// TIA Portal V17 export
// export: Created 2025-06-20T10:23:48.7607854Z, ExportSetting WithDefaults, DisplayName Totally Integrated Automation Portal, DisplayVersion V17 Update 8, DisplayName TIA Portal Openness, DisplayVersion V17 Update 8, DisplayName TIA Portal Version Control Interface, DisplayVersion V17, DisplayName SINAMICS Startdrive Advanced, DisplayVersion V17 SP2, DisplayName SINAMICS Startdrive G110M, G120, G120C, G120D, G120P, G115D, DisplayVersion V17 SP2, DisplayName SINAMICS Startdrive G130, G150, S120, S150, SINAMICS MV, S210, DisplayVersion V17 SP2, DisplayName STEP 7 Professional, DisplayVersion V17 Update 8, DisplayName SINUMERIK ONE STEP 7 Toolbox, DisplayVersion V17 Update 12, DisplayName SINUMERIK ONE PLC Basic Program Plus, DisplayVersion V17 Update 12, DisplayName SINUMERIK 840D sl STEP 7 Toolbox, DisplayVersion V17 Update 12, DisplayName STEP 7 Safety, DisplayVersion V17 Update 6, DisplayName WinCC Advanced, DisplayVersion V17 Update 8
FUNCTION "FC441_MACHINE_POWDER_ALARM_DECODING" : Void   // FC441, LAD
{ S7_Optimized_Access := 'FALSE' }
AUTHOR : ETXETAR
VERSION : 1.0
// stored: AutoNumber false, IsIECCheckEnabled false, SetENOAutomatically false, UDAEnableTagReadback false
   VAR_TEMP
      RST_ALARMS_1 : Bool;   // RESET ALARMS 1
      RST_ALARMS_2 : Bool;   // RESET ALARMS 2
      ZERO : Int;   // ZERO
      RET_VAL_1 : Int;   // RET VALUE
   END_VAR
   VAR CONSTANT
      FC_CONSTANT : Int := 440;
   END_VAR
   VAR_TEMP   // added for the SCL form of the ladder/FBD networks
      _w1 : Bool;
      _w2 : Bool;
      _w3 : Bool;
   END_VAR
BEGIN

REGION Network 1: ZERO
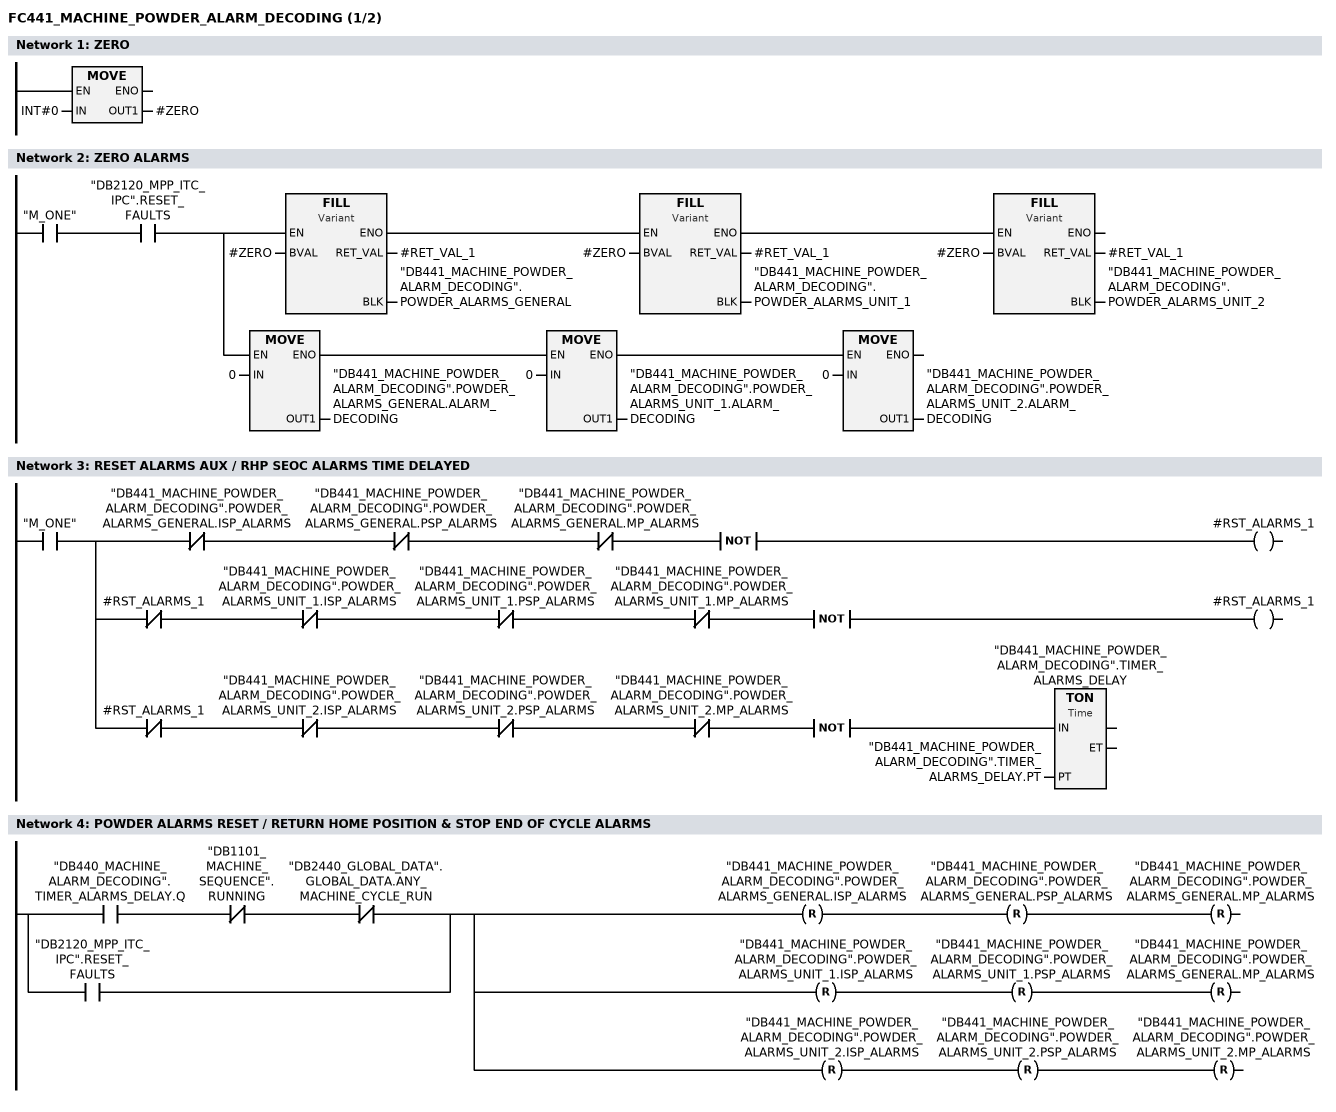
   RUNG wire#powerrail
      { S7_GenerateENO := "TRUE" } Move(in := INT#0, out1 => #ZERO)
   END_RUNG
   // the same network as SCL:
   #ZERO := INT#0;
END_REGION

REGION Network 2: ZERO ALARMS
   RUNG wire#powerrail
      Contact( "M_ONE" )
      Contact( "DB2120_MPP_ITC_IPC".RESET_FAULTS )
      wire#w1
      { S7_Templates := "ptr_type := Variant" } FILL(BVAL := #ZERO, RET_VAL => #RET_VAL_1, BLK => "DB441_MACHINE_POWDER_ALARM_DECODING".POWDER_ALARMS_GENERAL)
      { S7_Templates := "ptr_type := Variant" } FILL(BVAL := #ZERO, RET_VAL => #RET_VAL_1, BLK => "DB441_MACHINE_POWDER_ALARM_DECODING".POWDER_ALARMS_UNIT_1)
      { S7_Templates := "ptr_type := Variant" } FILL(BVAL := #ZERO, RET_VAL => #RET_VAL_1, BLK => "DB441_MACHINE_POWDER_ALARM_DECODING".POWDER_ALARMS_UNIT_2)
   END_RUNG
   RUNG wire#w1
      { S7_GenerateENO := "TRUE" } Move(in := 0, out1 => "DB441_MACHINE_POWDER_ALARM_DECODING".POWDER_ALARMS_GENERAL.ALARM_DECODING)
      { S7_GenerateENO := "TRUE" } Move(in := 0, out1 => "DB441_MACHINE_POWDER_ALARM_DECODING".POWDER_ALARMS_UNIT_1.ALARM_DECODING)
      { S7_GenerateENO := "TRUE" } Move(in := 0, out1 => "DB441_MACHINE_POWDER_ALARM_DECODING".POWDER_ALARMS_UNIT_2.ALARM_DECODING)
   END_RUNG
   // the same network as SCL:
   // ENO of a box is taken as its EN; it also drops when the box reports an error
   #_w2 := "M_ONE" AND "DB2120_MPP_ITC_IPC".RESET_FAULTS;
   #RET_VAL_1 := FILL(EN := "M_ONE" AND "DB2120_MPP_ITC_IPC".RESET_FAULTS,
                      BVAL := #ZERO,
                      BLK => "DB441_MACHINE_POWDER_ALARM_DECODING".POWDER_ALARMS_GENERAL,
                      ENO => #_w1);
   #RET_VAL_1 := FILL(EN := #_w1,
                      BVAL := #ZERO,
                      BLK => "DB441_MACHINE_POWDER_ALARM_DECODING".POWDER_ALARMS_UNIT_1,
                      ENO => #_w3);
   IF #_w3 THEN
       #RET_VAL_1 := FILL(BVAL := #ZERO, BLK => "DB441_MACHINE_POWDER_ALARM_DECODING".POWDER_ALARMS_UNIT_2);
   END_IF;
   IF #_w2 THEN
       "DB441_MACHINE_POWDER_ALARM_DECODING".POWDER_ALARMS_GENERAL.ALARM_DECODING := 0;
       "DB441_MACHINE_POWDER_ALARM_DECODING".POWDER_ALARMS_UNIT_1.ALARM_DECODING := 0;
       "DB441_MACHINE_POWDER_ALARM_DECODING".POWDER_ALARMS_UNIT_2.ALARM_DECODING := 0;
   END_IF;
END_REGION

REGION Network 3: RESET ALARMS AUX / RHP SEOC ALARMS TIME DELAYED
   RUNG wire#powerrail
      Contact( "M_ONE" )
      wire#w1
      I_Contact( "DB441_MACHINE_POWDER_ALARM_DECODING".POWDER_ALARMS_GENERAL.ISP_ALARMS )
      I_Contact( "DB441_MACHINE_POWDER_ALARM_DECODING".POWDER_ALARMS_GENERAL.PSP_ALARMS )
      I_Contact( "DB441_MACHINE_POWDER_ALARM_DECODING".POWDER_ALARMS_GENERAL.MP_ALARMS )
      Not()
      Coil( #RST_ALARMS_1 )
   END_RUNG
   RUNG wire#w1
      I_Contact( #RST_ALARMS_1 )
      I_Contact( "DB441_MACHINE_POWDER_ALARM_DECODING".POWDER_ALARMS_UNIT_1.ISP_ALARMS )
      I_Contact( "DB441_MACHINE_POWDER_ALARM_DECODING".POWDER_ALARMS_UNIT_1.PSP_ALARMS )
      I_Contact( "DB441_MACHINE_POWDER_ALARM_DECODING".POWDER_ALARMS_UNIT_1.MP_ALARMS )
      Not()
      Coil( #RST_ALARMS_1 )
   END_RUNG
   RUNG wire#w1
      I_Contact( #RST_ALARMS_1 )
      I_Contact( "DB441_MACHINE_POWDER_ALARM_DECODING".POWDER_ALARMS_UNIT_2.ISP_ALARMS )
      I_Contact( "DB441_MACHINE_POWDER_ALARM_DECODING".POWDER_ALARMS_UNIT_2.PSP_ALARMS )
      I_Contact( "DB441_MACHINE_POWDER_ALARM_DECODING".POWDER_ALARMS_UNIT_2.MP_ALARMS )
      Not()
      { S7_Templates := "time_type := Time" } "DB441_MACHINE_POWDER_ALARM_DECODING".TIMER_ALARMS_DELAY.TON(pt := "DB441_MACHINE_POWDER_ALARM_DECODING".TIMER_ALARMS_DELAY.PT, et =>)
   END_RUNG
   // the same network as SCL:
   #RST_ALARMS_1 := NOT ("M_ONE" AND NOT "DB441_MACHINE_POWDER_ALARM_DECODING".POWDER_ALARMS_GENERAL.ISP_ALARMS AND NOT "DB441_MACHINE_POWDER_ALARM_DECODING".POWDER_ALARMS_GENERAL.PSP_ALARMS AND NOT "DB441_MACHINE_POWDER_ALARM_DECODING".POWDER_ALARMS_GENERAL.MP_ALARMS);
   #RST_ALARMS_1 := NOT ("M_ONE" AND NOT #RST_ALARMS_1 AND NOT "DB441_MACHINE_POWDER_ALARM_DECODING".POWDER_ALARMS_UNIT_1.ISP_ALARMS AND NOT "DB441_MACHINE_POWDER_ALARM_DECODING".POWDER_ALARMS_UNIT_1.PSP_ALARMS AND NOT "DB441_MACHINE_POWDER_ALARM_DECODING".POWDER_ALARMS_UNIT_1.MP_ALARMS);
   "DB441_MACHINE_POWDER_ALARM_DECODING".TIMER_ALARMS_DELAY.TON(IN := NOT ("M_ONE" AND NOT #RST_ALARMS_1 AND NOT "DB441_MACHINE_POWDER_ALARM_DECODING".POWDER_ALARMS_UNIT_2.ISP_ALARMS AND NOT "DB441_MACHINE_POWDER_ALARM_DECODING".POWDER_ALARMS_UNIT_2.PSP_ALARMS AND NOT "DB441_MACHINE_POWDER_ALARM_DECODING".POWDER_ALARMS_UNIT_2.MP_ALARMS),
                           PT := "DB441_MACHINE_POWDER_ALARM_DECODING".TIMER_ALARMS_DELAY.PT);
END_REGION

REGION Network 4: POWDER ALARMS RESET / RETURN HOME POSITION & STOP END OF CYCLE ALARMS
   RUNG wire#powerrail
      Contact( "DB440_MACHINE_ALARM_DECODING".TIMER_ALARMS_DELAY.Q )
      I_Contact( "DB1101_MACHINE_SEQUENCE".RUNNING )
      I_Contact( "DB2440_GLOBAL_DATA".GLOBAL_DATA.ANY_MACHINE_CYCLE_RUN )
      wire#w1
      R_Coil( "DB441_MACHINE_POWDER_ALARM_DECODING".POWDER_ALARMS_GENERAL.ISP_ALARMS )
      R_Coil( "DB441_MACHINE_POWDER_ALARM_DECODING".POWDER_ALARMS_GENERAL.PSP_ALARMS )
      R_Coil( "DB441_MACHINE_POWDER_ALARM_DECODING".POWDER_ALARMS_GENERAL.MP_ALARMS )
   END_RUNG
   RUNG wire#powerrail
      Contact( "DB2120_MPP_ITC_IPC".RESET_FAULTS )
   END_RUNG wire#w1
   RUNG wire#w1
      R_Coil( "DB441_MACHINE_POWDER_ALARM_DECODING".POWDER_ALARMS_UNIT_1.ISP_ALARMS )
      R_Coil( "DB441_MACHINE_POWDER_ALARM_DECODING".POWDER_ALARMS_UNIT_1.PSP_ALARMS )
      R_Coil( "DB441_MACHINE_POWDER_ALARM_DECODING".POWDER_ALARMS_GENERAL.MP_ALARMS )
   END_RUNG
   RUNG wire#w1
      R_Coil( "DB441_MACHINE_POWDER_ALARM_DECODING".POWDER_ALARMS_UNIT_2.ISP_ALARMS )
      R_Coil( "DB441_MACHINE_POWDER_ALARM_DECODING".POWDER_ALARMS_UNIT_2.PSP_ALARMS )
      R_Coil( "DB441_MACHINE_POWDER_ALARM_DECODING".POWDER_ALARMS_UNIT_2.MP_ALARMS )
   END_RUNG
   // the same network as SCL:
   IF ("DB440_MACHINE_ALARM_DECODING".TIMER_ALARMS_DELAY.Q AND NOT "DB1101_MACHINE_SEQUENCE".RUNNING AND NOT "DB2440_GLOBAL_DATA".GLOBAL_DATA.ANY_MACHINE_CYCLE_RUN) OR "DB2120_MPP_ITC_IPC".RESET_FAULTS THEN
       "DB441_MACHINE_POWDER_ALARM_DECODING".POWDER_ALARMS_GENERAL.ISP_ALARMS := FALSE;
       "DB441_MACHINE_POWDER_ALARM_DECODING".POWDER_ALARMS_GENERAL.PSP_ALARMS := FALSE;
       "DB441_MACHINE_POWDER_ALARM_DECODING".POWDER_ALARMS_GENERAL.MP_ALARMS := FALSE;
       "DB441_MACHINE_POWDER_ALARM_DECODING".POWDER_ALARMS_UNIT_1.ISP_ALARMS := FALSE;
       "DB441_MACHINE_POWDER_ALARM_DECODING".POWDER_ALARMS_UNIT_1.PSP_ALARMS := FALSE;
       "DB441_MACHINE_POWDER_ALARM_DECODING".POWDER_ALARMS_GENERAL.MP_ALARMS := FALSE;
       "DB441_MACHINE_POWDER_ALARM_DECODING".POWDER_ALARMS_UNIT_2.ISP_ALARMS := FALSE;
       "DB441_MACHINE_POWDER_ALARM_DECODING".POWDER_ALARMS_UNIT_2.PSP_ALARMS := FALSE;
       "DB441_MACHINE_POWDER_ALARM_DECODING".POWDER_ALARMS_UNIT_2.MP_ALARMS := FALSE;
   END_IF;
END_REGION

REGION Network 5: <<<<<<<<<<<<<<<<<<<< ALARMS BY UNITS >>>>>>>>>>>>>>>>>>>>
END_REGION

REGION Network 6: ALARMS
   // Cada uno de estos iria ordenadamente en las señales del interlock con polvo / Stations Faulted
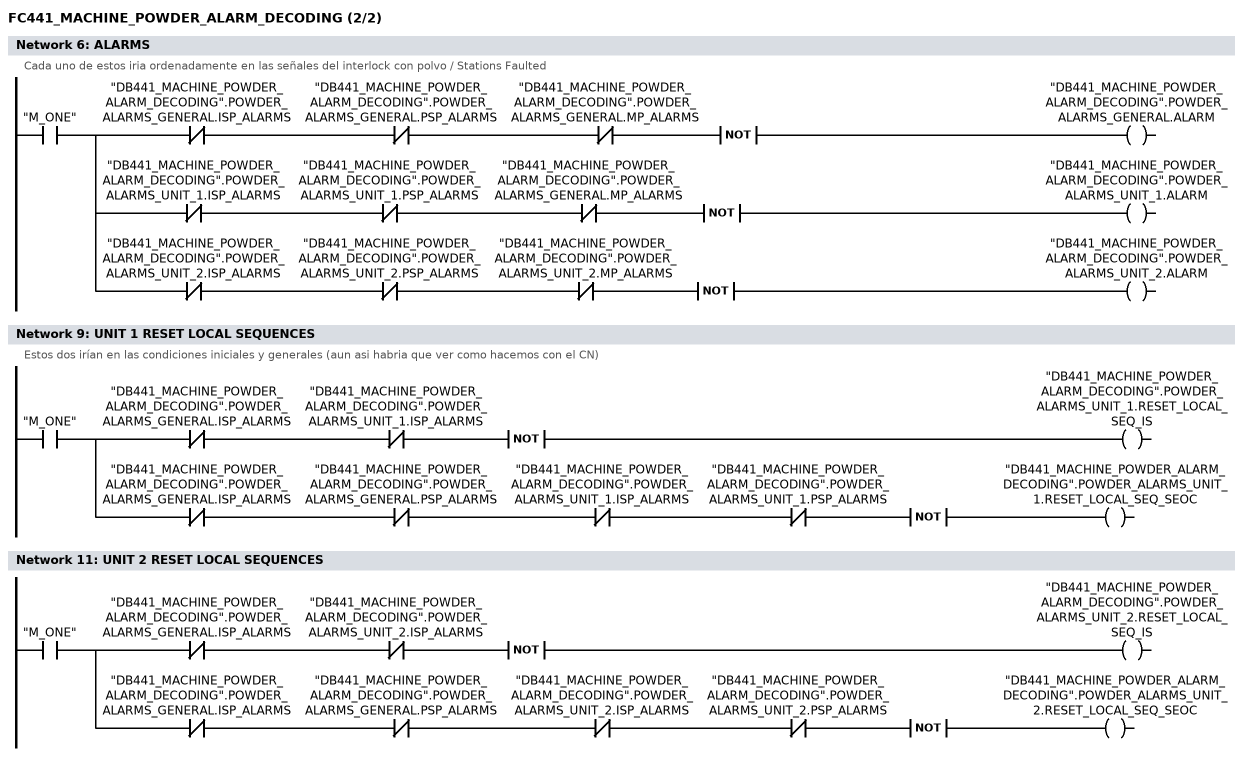
   RUNG wire#powerrail
      Contact( "M_ONE" )
      wire#w1
      I_Contact( "DB441_MACHINE_POWDER_ALARM_DECODING".POWDER_ALARMS_GENERAL.ISP_ALARMS )
      I_Contact( "DB441_MACHINE_POWDER_ALARM_DECODING".POWDER_ALARMS_GENERAL.PSP_ALARMS )
      I_Contact( "DB441_MACHINE_POWDER_ALARM_DECODING".POWDER_ALARMS_GENERAL.MP_ALARMS )
      Not()
      Coil( "DB441_MACHINE_POWDER_ALARM_DECODING".POWDER_ALARMS_GENERAL.ALARM )
   END_RUNG
   RUNG wire#w1
      I_Contact( "DB441_MACHINE_POWDER_ALARM_DECODING".POWDER_ALARMS_UNIT_1.ISP_ALARMS )
      I_Contact( "DB441_MACHINE_POWDER_ALARM_DECODING".POWDER_ALARMS_UNIT_1.PSP_ALARMS )
      I_Contact( "DB441_MACHINE_POWDER_ALARM_DECODING".POWDER_ALARMS_GENERAL.MP_ALARMS )
      Not()
      Coil( "DB441_MACHINE_POWDER_ALARM_DECODING".POWDER_ALARMS_UNIT_1.ALARM )
   END_RUNG
   RUNG wire#w1
      I_Contact( "DB441_MACHINE_POWDER_ALARM_DECODING".POWDER_ALARMS_UNIT_2.ISP_ALARMS )
      I_Contact( "DB441_MACHINE_POWDER_ALARM_DECODING".POWDER_ALARMS_UNIT_2.PSP_ALARMS )
      I_Contact( "DB441_MACHINE_POWDER_ALARM_DECODING".POWDER_ALARMS_UNIT_2.MP_ALARMS )
      Not()
      Coil( "DB441_MACHINE_POWDER_ALARM_DECODING".POWDER_ALARMS_UNIT_2.ALARM )
   END_RUNG
   // the same network as SCL:
   "DB441_MACHINE_POWDER_ALARM_DECODING".POWDER_ALARMS_GENERAL.ALARM := NOT ("M_ONE" AND NOT "DB441_MACHINE_POWDER_ALARM_DECODING".POWDER_ALARMS_GENERAL.ISP_ALARMS AND NOT "DB441_MACHINE_POWDER_ALARM_DECODING".POWDER_ALARMS_GENERAL.PSP_ALARMS AND NOT "DB441_MACHINE_POWDER_ALARM_DECODING".POWDER_ALARMS_GENERAL.MP_ALARMS);
   "DB441_MACHINE_POWDER_ALARM_DECODING".POWDER_ALARMS_UNIT_1.ALARM := NOT ("M_ONE" AND NOT "DB441_MACHINE_POWDER_ALARM_DECODING".POWDER_ALARMS_UNIT_1.ISP_ALARMS AND NOT "DB441_MACHINE_POWDER_ALARM_DECODING".POWDER_ALARMS_UNIT_1.PSP_ALARMS AND NOT "DB441_MACHINE_POWDER_ALARM_DECODING".POWDER_ALARMS_GENERAL.MP_ALARMS);
   "DB441_MACHINE_POWDER_ALARM_DECODING".POWDER_ALARMS_UNIT_2.ALARM := NOT ("M_ONE" AND NOT "DB441_MACHINE_POWDER_ALARM_DECODING".POWDER_ALARMS_UNIT_2.ISP_ALARMS AND NOT "DB441_MACHINE_POWDER_ALARM_DECODING".POWDER_ALARMS_UNIT_2.PSP_ALARMS AND NOT "DB441_MACHINE_POWDER_ALARM_DECODING".POWDER_ALARMS_UNIT_2.MP_ALARMS);
END_REGION

REGION Network 7: <<<<<<<<<<<<<<<<<<<< ALARMS BY UNIT >>>>>>>>>>>>>>>>>>>>
END_REGION

REGION Network 8: <<<<<<<<<<<<<<<<<<<<<<<< UNIT 1 >>>>>>>>>>>>>>>>>>>>>>>>
END_REGION

REGION Network 9: UNIT 1 RESET LOCAL SEQUENCES
   // Estos dos irían en las condiciones iniciales y generales (aun asi habria que ver como hacemos con el CN)
   RUNG wire#powerrail
      Contact( "M_ONE" )
      wire#w1
      I_Contact( "DB441_MACHINE_POWDER_ALARM_DECODING".POWDER_ALARMS_GENERAL.ISP_ALARMS )
      I_Contact( "DB441_MACHINE_POWDER_ALARM_DECODING".POWDER_ALARMS_UNIT_1.ISP_ALARMS )
      Not()
      Coil( "DB441_MACHINE_POWDER_ALARM_DECODING".POWDER_ALARMS_UNIT_1.RESET_LOCAL_SEQ_IS )
   END_RUNG
   RUNG wire#w1
      I_Contact( "DB441_MACHINE_POWDER_ALARM_DECODING".POWDER_ALARMS_GENERAL.ISP_ALARMS )
      I_Contact( "DB441_MACHINE_POWDER_ALARM_DECODING".POWDER_ALARMS_GENERAL.PSP_ALARMS )
      I_Contact( "DB441_MACHINE_POWDER_ALARM_DECODING".POWDER_ALARMS_UNIT_1.ISP_ALARMS )
      I_Contact( "DB441_MACHINE_POWDER_ALARM_DECODING".POWDER_ALARMS_UNIT_1.PSP_ALARMS )
      Not()
      Coil( "DB441_MACHINE_POWDER_ALARM_DECODING".POWDER_ALARMS_UNIT_1.RESET_LOCAL_SEQ_SEOC )
   END_RUNG
   // the same network as SCL:
   "DB441_MACHINE_POWDER_ALARM_DECODING".POWDER_ALARMS_UNIT_1.RESET_LOCAL_SEQ_IS := NOT ("M_ONE" AND NOT "DB441_MACHINE_POWDER_ALARM_DECODING".POWDER_ALARMS_GENERAL.ISP_ALARMS AND NOT "DB441_MACHINE_POWDER_ALARM_DECODING".POWDER_ALARMS_UNIT_1.ISP_ALARMS);
   "DB441_MACHINE_POWDER_ALARM_DECODING".POWDER_ALARMS_UNIT_1.RESET_LOCAL_SEQ_SEOC := NOT ("M_ONE" AND NOT "DB441_MACHINE_POWDER_ALARM_DECODING".POWDER_ALARMS_GENERAL.ISP_ALARMS AND NOT "DB441_MACHINE_POWDER_ALARM_DECODING".POWDER_ALARMS_GENERAL.PSP_ALARMS AND NOT "DB441_MACHINE_POWDER_ALARM_DECODING".POWDER_ALARMS_UNIT_1.ISP_ALARMS AND NOT "DB441_MACHINE_POWDER_ALARM_DECODING".POWDER_ALARMS_UNIT_1.PSP_ALARMS);
END_REGION

REGION Network 10: <<<<<<<<<<<<<<<<<<<<<<<< UNIT 2 >>>>>>>>>>>>>>>>>>>>>>>>
END_REGION

REGION Network 11: UNIT 2 RESET LOCAL SEQUENCES
   RUNG wire#powerrail
      Contact( "M_ONE" )
      wire#w1
      I_Contact( "DB441_MACHINE_POWDER_ALARM_DECODING".POWDER_ALARMS_GENERAL.ISP_ALARMS )
      I_Contact( "DB441_MACHINE_POWDER_ALARM_DECODING".POWDER_ALARMS_UNIT_2.ISP_ALARMS )
      Not()
      Coil( "DB441_MACHINE_POWDER_ALARM_DECODING".POWDER_ALARMS_UNIT_2.RESET_LOCAL_SEQ_IS )
   END_RUNG
   RUNG wire#w1
      I_Contact( "DB441_MACHINE_POWDER_ALARM_DECODING".POWDER_ALARMS_GENERAL.ISP_ALARMS )
      I_Contact( "DB441_MACHINE_POWDER_ALARM_DECODING".POWDER_ALARMS_GENERAL.PSP_ALARMS )
      I_Contact( "DB441_MACHINE_POWDER_ALARM_DECODING".POWDER_ALARMS_UNIT_2.ISP_ALARMS )
      I_Contact( "DB441_MACHINE_POWDER_ALARM_DECODING".POWDER_ALARMS_UNIT_2.PSP_ALARMS )
      Not()
      Coil( "DB441_MACHINE_POWDER_ALARM_DECODING".POWDER_ALARMS_UNIT_2.RESET_LOCAL_SEQ_SEOC )
   END_RUNG
   // the same network as SCL:
   "DB441_MACHINE_POWDER_ALARM_DECODING".POWDER_ALARMS_UNIT_2.RESET_LOCAL_SEQ_IS := NOT ("M_ONE" AND NOT "DB441_MACHINE_POWDER_ALARM_DECODING".POWDER_ALARMS_GENERAL.ISP_ALARMS AND NOT "DB441_MACHINE_POWDER_ALARM_DECODING".POWDER_ALARMS_UNIT_2.ISP_ALARMS);
   "DB441_MACHINE_POWDER_ALARM_DECODING".POWDER_ALARMS_UNIT_2.RESET_LOCAL_SEQ_SEOC := NOT ("M_ONE" AND NOT "DB441_MACHINE_POWDER_ALARM_DECODING".POWDER_ALARMS_GENERAL.ISP_ALARMS AND NOT "DB441_MACHINE_POWDER_ALARM_DECODING".POWDER_ALARMS_GENERAL.PSP_ALARMS AND NOT "DB441_MACHINE_POWDER_ALARM_DECODING".POWDER_ALARMS_UNIT_2.ISP_ALARMS AND NOT "DB441_MACHINE_POWDER_ALARM_DECODING".POWDER_ALARMS_UNIT_2.PSP_ALARMS);
END_REGION
END_FUNCTION
